// TIA Portal V16 export
// export: Created 2021-04-06T19:52:16.5127396Z, ExportSetting WithDefaults, DisplayName Totally Integrated Automation Portal, DisplayVersion V16, DisplayName TIA Portal Version Control Interface, DisplayVersion V16, DisplayName TIA Portal Openness, DisplayVersion V16, DisplayName STEP 7 Professional, DisplayVersion V16, DisplayName STEP 7 Safety, DisplayVersion V16, DisplayName WinCC Unified SCADA Engineering System, DisplayVersion V16
FUNCTION_BLOCK "workVibroTable_AM"   // FB7, LAD
TITLE = Управление вибростолами
{ S7_Optimized_Access := 'TRUE' }
VERSION : 0.1
// На основе массивов готовности бункеров к сортировке решаем работать столу или нет
// stored: AutoNumber true, IsIECCheckEnabled false, IsRetainMemResEnabled false, MemoryReserve 100, SetENOAutomatically false, UDAEnableTagReadback false
   VAR_INPUT
      enableWork : Bool;
      alarmStop : Bool;
      arrayReadyWeightBunker : Array[0..12] of Bool;
   END_VAR
   VAR_OUTPUT
      vibroTable : Array[0..2] of Bool;
   END_VAR
   VAR
      tmpValueReadyWeight : Array[0..2] of Bool;
   END_VAR
   VAR_TEMP
      i : SInt;
   END_VAR
BEGIN

REGION Network 1 (SCL)
   //в массиве arrayReadyWeightBunker храняться состояния готовности веса в бункерах

   IF #enableWork AND NOT(#alarmStop) THEN
       #tmpValueReadyWeight[1] := true;
       #tmpValueReadyWeight[2] := true;
       #i := 0;
       FOR #i := 1 TO 6 DO
           #tmpValueReadyWeight[1] := #tmpValueReadyWeight[1] AND #arrayReadyWeightBunker[#i];
           #tmpValueReadyWeight[2] := #tmpValueReadyWeight[2] AND #arrayReadyWeightBunker[#i + 6];
       END_FOR;
       #i := 0;
       FOR #i := 1 TO 2 DO
           IF NOT (#tmpValueReadyWeight[#i]) THEN //#tmpValueReadyWeight=0 если хотябы один бункер не готов
               #vibroTable[#i] := true;
           ELSE
               #vibroTable[#i] := false;
           END_IF;
       END_FOR;
   ELSE
       #vibroTable[1] := false;
       #vibroTable[2] := false;
   END_IF;
END_REGION
END_FUNCTION_BLOCK
